// TIA Portal V17 export
// export: Created 2023-12-22T15:05:29.7602113Z, ExportSetting WithDefaults, DisplayName Totally Integrated Automation Portal, DisplayVersion V17, DisplayName TIA Portal Openness, DisplayVersion V17, DisplayName TIA Portal Version Control Interface, DisplayVersion V17, DisplayName STEP 7 Professional, DisplayVersion V17, DisplayName STEP 7 Safety, DisplayVersion V17, DisplayName WinCC Advanced, DisplayVersion V17
DATA_BLOCK "DOx_1_DB"   // DB210
VERSION : 0.1
// stored: AutoNumber false, DBAccessibleFromOPCUA true, InstanceOfName DOx_1, InstanceOfType FB
"DOx_1"
   // VAR RETAIN
   //    EZ_1_Alarm_Stop { S7_SetPoint := 'True'} : "DO_ex";
   //    Red_Signal { S7_SetPoint := 'True'} : "DO_ex";
   //    KC_1_Start { S7_SetPoint := 'True'} : "DO_ex";
   //    KC_2_Start { S7_SetPoint := 'True'} : "DO_ex";
   //    command_5 { S7_SetPoint := 'True'} : "DO_ex";
   //    command_6 { S7_SetPoint := 'True'} : "DO_ex";
   //    command_7 { S7_SetPoint := 'True'} : "DO_ex";
   //    command_8 { S7_SetPoint := 'True'} : "DO_ex";
   //    command_9 { S7_SetPoint := 'True'} : "DO_ex";
   //    command_10 { S7_SetPoint := 'True'} : "DO_ex";
   //    command_11 { S7_SetPoint := 'True'} : "DO_ex";
   //    command_12 { S7_SetPoint := 'True'} : "DO_ex";
   //    Time_DTL { S7_SetPoint := 'True'} : DTL := DTL#2012-01-01-20:29:23.799879;
   // END_VAR
BEGIN
   EZ_1_Alarm_Stop.Use.Inverse := TRUE;
   EZ_1_Alarm_Stop.Use.Indirect := TRUE;
   EZ_1_Alarm_Stop.Use.Impulse := FALSE;
   EZ_1_Alarm_Stop.ADDR_Byte := 0;
   EZ_1_Alarm_Stop.ADDR_Bit := 1;
   EZ_1_Alarm_Stop.T_Impulse.SP := 16#02;
   Red_Signal.Use.Inverse := FALSE;
   Red_Signal.Use.Indirect := TRUE;
   Red_Signal.Use.Impulse := FALSE;
   Red_Signal.ADDR_Byte := 0;
   Red_Signal.ADDR_Bit := 6;
   Red_Signal.T_Impulse.SP := 16#02;
   KC_1_Start.Use.Inverse := FALSE;
   KC_1_Start.Use.Indirect := TRUE;
   KC_1_Start.Use.Impulse := FALSE;
   KC_1_Start.ADDR_Byte := 0;
   KC_1_Start.ADDR_Bit := 4;
   KC_1_Start.T_Impulse.SP := 16#02;
   KC_2_Start.Use.Inverse := FALSE;
   KC_2_Start.Use.Indirect := TRUE;
   KC_2_Start.Use.Impulse := FALSE;
   KC_2_Start.ADDR_Byte := 0;
   KC_2_Start.ADDR_Bit := 5;
   KC_2_Start.T_Impulse.SP := 16#02;
   command_5.Use.Inverse := FALSE;
   command_5.Use.Indirect := TRUE;
   command_5.Use.Impulse := FALSE;
   command_5.ADDR_Byte := 0;
   command_5.ADDR_Bit := 9;
   command_5.T_Impulse.SP := 16#02;
   command_6.Use.Inverse := FALSE;
   command_6.Use.Indirect := TRUE;
   command_6.Use.Impulse := FALSE;
   command_6.ADDR_Byte := 0;
   command_6.ADDR_Bit := 9;
   command_6.T_Impulse.SP := 16#02;
   command_7.Use.Inverse := FALSE;
   command_7.Use.Indirect := TRUE;
   command_7.Use.Impulse := FALSE;
   command_7.ADDR_Byte := 0;
   command_7.ADDR_Bit := 9;
   command_7.T_Impulse.SP := 16#02;
   command_8.Use.Inverse := FALSE;
   command_8.Use.Indirect := TRUE;
   command_8.Use.Impulse := FALSE;
   command_8.ADDR_Byte := 0;
   command_8.ADDR_Bit := 9;
   command_8.T_Impulse.SP := 16#02;
   command_9.Use.Inverse := FALSE;
   command_9.Use.Indirect := TRUE;
   command_9.Use.Impulse := FALSE;
   command_9.ADDR_Byte := 0;
   command_9.ADDR_Bit := 9;
   command_9.T_Impulse.SP := 16#02;
   command_10.Use.Inverse := FALSE;
   command_10.Use.Indirect := TRUE;
   command_10.Use.Impulse := FALSE;
   command_10.ADDR_Byte := 0;
   command_10.ADDR_Bit := 9;
   command_10.T_Impulse.SP := 16#02;
   command_11.Use.Inverse := FALSE;
   command_11.Use.Indirect := TRUE;
   command_11.Use.Impulse := FALSE;
   command_11.ADDR_Byte := 0;
   command_11.ADDR_Bit := 9;
   command_11.T_Impulse.SP := 16#02;
   command_12.Use.Inverse := FALSE;
   command_12.Use.Indirect := TRUE;
   command_12.Use.Impulse := FALSE;
   command_12.ADDR_Byte := 0;
   command_12.ADDR_Bit := 9;
   command_12.T_Impulse.SP := 16#02;
END_DATA_BLOCK
